ABB RobotStudio station: Prova_1.rsstnx

Station Prova_1 (saved by RobotStudio 22.3.10190.2)
Controller CRB15000_5_95
  mechanical unit ROB_1: CRB15000_5_95__02, 6 joints, base frame (0, 0, 0) mm
Layout (positions relative to the parent item):
  - CRB15000_5_95__02 [mechanism, from Robots\CRB15000_5_95__02.rslib] at (0, 0, 0) mm; joint values [0.736, 0.4822, -0.796, -0.633, 2.2606, 1.9887] (rad or m)
  - GeoUteCollisione [part] at (531.89, 378.91, 808.53) mm, rotated rx 180 ry 38 rz 90 deg, size 219.3 x 84 x 110.4 mm
  - Table [part] at (306.89, 137.59, 0) mm, size 450 x 350 x 308 mm
  - Parte_1 [part] at (331.89, 262.59, 308) mm, size 200 x 200 x 300 mm
  - MyNewTool [mechanism] at (531.89, 378.91, 808.53) mm, rotated rx 180 ry 38 rz 90 deg
      links: Dummy
  - MyTool [mechanism, from Training Objects\myTool.rslib] at (531.89, 378.91, 808.53) mm, rotated rx 180 ry 38 rz 90 deg
Attachment: GeoUteCollisione is attached to CRB15000_5_95__02 / Link6
Attachment: MyNewTool is attached to CRB15000_5_95__02 / Link6
Attachment: MyTool is attached to CRB15000_5_95__02 / Link6
Targets, tools, work objects and paths stored in the station, written as RAPID:
! task T_ROB1
MODULE CalibData
  PERS wobjdata Workobject_1:=[FALSE,TRUE,"",[[331.886,262.587,608],[1,0,0,0]],[[0,0,0],[1,0,0,0]]];
  PERS tooldata MyTool:=[TRUE,[[31.792631019,0,229.638935148],[0.945518576,0,0.325568154,0]],[1,[0,0,1],[1,0,0,0],0,0,0]];
ENDMODULE

! task T_ROB1
MODULE Module1
  CONST robtarget Target_10:=[[-0.000096788,0,-0.000128503],[0,-0.707106781,0.707106781,0],[0,0,0,0],[9E+09,9E+09,9E+09,9E+09,9E+09,9E+09]];
  CONST robtarget Target_20:=[[199.999903212,0,-0.000128503],[0,0.707106781,0.707106781,0],[0,0,1,0],[9E+09,9E+09,9E+09,9E+09,9E+09,9E+09]];
  PROC Path_10()
    MoveJ Target_10,v1000,z100,MyTool\WObj:=Workobject_1;
    MoveJ Target_20,v1000,z100,MyTool\WObj:=Workobject_1;
  ENDPROC
ENDMODULE

